FUNCTION_BLOCK Q_ObjSelectInput (* Command Select input object ( Part 6 - F.6 ) *)
  (* Standard: ISO 11783-6; Description: Copyright (c) 2022 HR Agrartechnik GmbH This program and the accompanying materials are made available under the terms of the Eclipse Public License 2.0 which is available at https://www.eclipse.org/legal/epl-2.0/ SPDX-License-Identifier: EPL-2.0 see Description Tab *)
  (* Version 1.0, 2022-07-08, Franz Höpfinger, HR Agrartechnik GmbH *)
  PACKAGE isobus::UT::Q;
  IMPORT isobus::UT::Q::const::IDs::ID_NULL;
  (* Documentation:
  Command Select input object ( Part 6 - F.6 )
   This command is used to force the selection of an input field object.
   Valid Object IDs
   A select input Object ID is valid if it falls within one of the following ISO 11783-6 ID ranges:
    - Key: 5000 – 5999
   - Button: 6000 – 6999
   - InputBooleanField: 7000 – 7999
   - InputStringField: 8000 – 8999
   - InputNumberField: 9000 – 9999
   - InputListField: 10000 – 10999
    ID_NULL (65535) is not a command target but can be used in INIT to deactivate the FB. Any ID outside these ranges is invalid for commanding.
   Activate / Deactivate
   The FB is deactivated by default. It becomes active when INIT provides a valid select input Object ID. Sending INIT with ID_NULL (65535) deactivates the FB again. This toggle can be repeated arbitrarily.
    - INIT + ID_NULL (65535): FB deactivated, STATUS="DEACTIVATED", s16result=VT_E_DEACTIVATED (-40)
   - INIT + valid select input ID: FB activated, STATUS="initialized", s16result=VT_E_NO_ERR (0). If a REQ was buffered before, it is executed immediately.
   - INIT + invalid ID: STATUS="ERROR: Invalid Object ID (not a select input object)", s16result=VT_E_INVALID_OBJECT_ID (-132)
    REQ Handling
    - REQ before any INIT: Buffered, STATUS="Buffered: INIT not yet completed", s16result=VT_E_NOT_READY (-131)
   - REQ while deactivated (INIT came with NULL or invalid ID): STATUS shows the actual deactivation reason, s16result=VT_E_DEACTIVATED (-40) or VT_E_INVALID_OBJECT_ID (-132)
   - REQ while active: Command sent to VT, result reflected in CNF
    param[in] {objectID, uint16_t}
   Object ID of input object. Use ID_NULL (65535) to deactivate the FB. Use a valid select input object ID to activate.
   param[in] {option, uint8_t}
   normal: 0xFF, for Version 4 also 0 possible
   Return Values (s16result):
   int16_t
    - VT_E_NO_ERR (0) - OK
   - VT_E_DEACTIVATED (-40) - FB deactivated (INIT received with ID_NULL)
   - VT_E_INVALID_OBJECT_ID (-132) - Object ID is invalid (not a select input object)
   - VT_E_NOT_READY (-131) - Buffered: INIT not yet completed
   - VT_E_OVERFLOW (-6) - buffer overflow
   - VT_E_NOACT (-8) - Command not possible in current state
   - VT_E_NO_INSTANCE (-21) - No VT client available
   - VT_E_ISO_INSTANCE_INVALID (-129) - Identifier for instance (connection) invalid
   - VT_E_NOT_ALIVE (-130) - Identifier for instance valid, but VT Dead.
    Instanz-Eindeutigkeit (Instance Uniqueness)
   Dieser Baustein erfordert Instanz-Eindeutigkeit bezüglich u16ObjId. Es darf im gesamten Programm nur eine Instanz von Q_ObjSelectInput für dieselbe Ziel-Objekt-ID existieren. Eine zweite Instanz auf dieselbe Objekt-ID wird bei INIT deaktiviert (STATUS = "This objID is already in use").
  *)
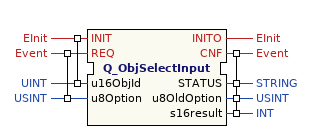
  EVENT_INPUT
    INIT : EInit WITH u16ObjId; (* Service Initialization *)
    REQ WITH u8Option; (* Service Request *)
  END_EVENT
  EVENT_OUTPUT
    INITO : EInit; (* Initialization Confirm *)
    CNF WITH STATUS, s16result, u8OldOption; (* Confirmation of Requested Service *)
  END_EVENT
  VAR_INPUT
    u16ObjId : UINT := ID_NULL; (* Object ID *)
    u8Option : USINT; (* normal: 0xFF, for Version 4 also 0 possible *)
  END_VAR
  VAR_OUTPUT
    STATUS : STRING; (* Service Status *)
    u8OldOption : USINT; (* Old normal: 0xFF, for Version 4 also 0 possible *)
    s16result : INT; (* retval see description *)
  END_VAR
END_FUNCTION_BLOCK
